Staubli VAL3: onF1Event.pgx

program onF1Event()
  local num i
begin
//  // look if the bButton is enable
  if bButton[0]
  popUpMsg("你按下了F1按键")
  endIf
end
